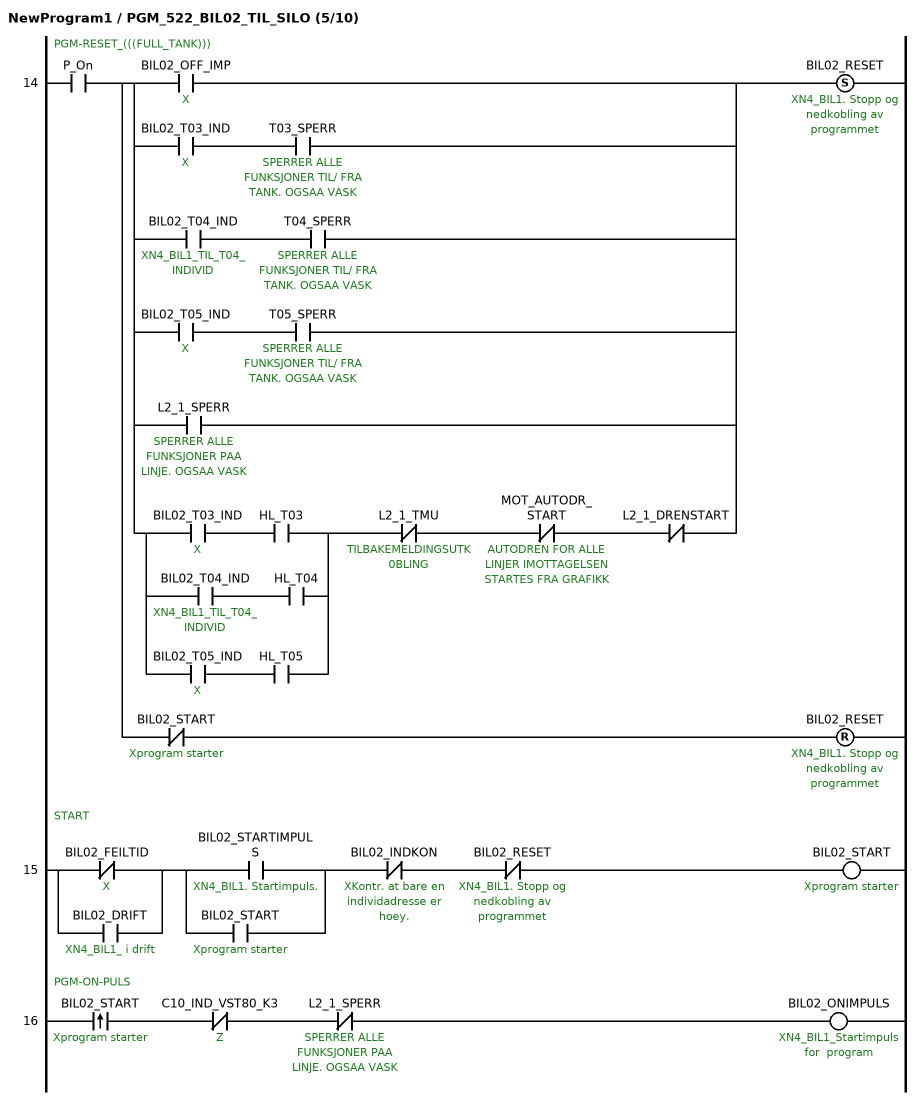
; [picture p624: NewProgram1 / PGM_522_BIL02_TIL_SILO, rungs 14-16]
; rung 14: PGM-RESET_(((FULL_TANK)))
LD P_On
OUT TR0
LD BIL02_OFF_IMP  ; X
LD BIL02_T03_IND  ; X
AND T03_SPERR  ; SPERRER ALLE FUNKSJONER TIL/ FRA TANK. OGSAA VASK
ORLD
LD BIL02_T04_IND  ; XN4_BIL1_TIL_T04_INDIVID
AND T04_SPERR  ; SPERRER ALLE FUNKSJONER TIL/ FRA TANK. OGSAA VASK
ORLD
LD BIL02_T05_IND  ; X
AND T05_SPERR  ; SPERRER ALLE FUNKSJONER TIL/ FRA TANK. OGSAA VASK
ORLD
OR L2_1_SPERR  ; SPERRER ALLE FUNKSJONER PAA LINJE. OGSAA VASK
LD BIL02_T03_IND  ; X
AND HL_T03
LD BIL02_T04_IND  ; XN4_BIL1_TIL_T04_INDIVID
AND HL_T04
ORLD
LD BIL02_T05_IND  ; X
AND HL_T05
ORLD
ANDNOT L2_1_TMU  ; TILBAKEMELDINGSUTK0BLING
ANDNOT MOT_AUTODR_START  ; AUTODREN FOR ALLE LINJER IMOTTAGELSEN STARTES FRA GRAFIKK
ANDNOT L2_1_DRENSTART
ORLD
ANDLD
SET BIL02_RESET  ; XN4_BIL1. Stopp og nedkobling av programmet
LD TR0
ANDNOT BIL02_START  ; Xprogram starter
RSET BIL02_RESET  ; XN4_BIL1. Stopp og nedkobling av programmet
; rung 15: START
LDNOT BIL02_FEILTID  ; X
OR BIL02_DRIFT  ; XN4_BIL1_ i drift
LD BIL02_STARTIMPULS  ; XN4_BIL1. Startimpuls.
OR BIL02_START  ; Xprogram starter
ANDLD
ANDNOT BIL02_INDKON  ; XKontr. at bare en individadresse er hoey.
ANDNOT BIL02_RESET  ; XN4_BIL1. Stopp og nedkobling av programmet
OUT BIL02_START  ; Xprogram starter
; rung 16: PGM-ON-PULS
@LD BIL02_START  ; Xprogram starter
ANDNOT C10_IND_VST80_K3  ; Z
ANDNOT L2_1_SPERR  ; SPERRER ALLE FUNKSJONER PAA LINJE. OGSAA VASK
OUT BIL02_ONIMPULS  ; XN4_BIL1_Startimpuls for  program

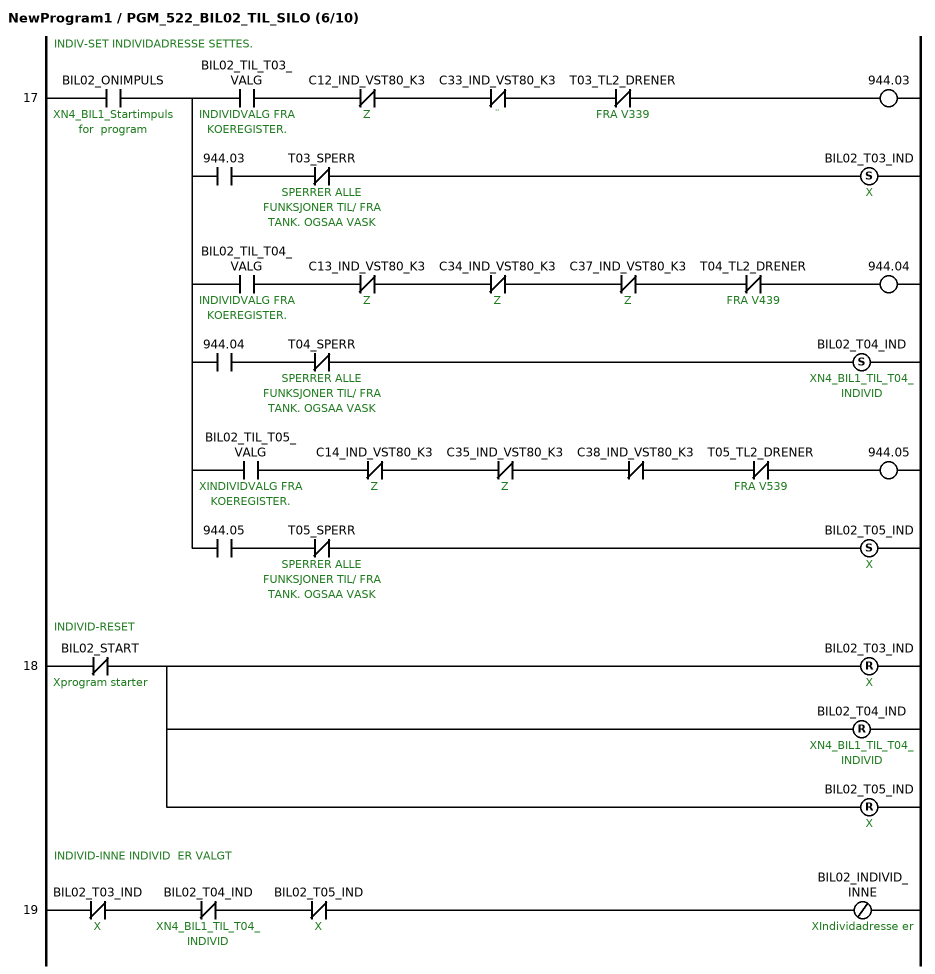
; rung 17: INDIV-SET INDIVIDADRESSE SETTES.
LD BIL02_ONIMPULS  ; XN4_BIL1_Startimpuls for  program
OUT TR0
AND BIL02_TIL_T03_VALG  ; INDIVIDVALG FRA KOEREGISTER.
ANDNOT C12_IND_VST80_K3  ; Z
ANDNOT C33_IND_VST80_K3  ; ¨
ANDNOT T03_TL2_DRENER  ; FRA V339
OUT 944.03
LD TR0
AND 944.03
ANDNOT T03_SPERR  ; SPERRER ALLE FUNKSJONER TIL/ FRA TANK. OGSAA VASK
SET BIL02_T03_IND  ; X
LD TR0
AND BIL02_TIL_T04_VALG  ; INDIVIDVALG FRA KOEREGISTER.
ANDNOT C13_IND_VST80_K3  ; Z
ANDNOT C34_IND_VST80_K3  ; Z
ANDNOT C37_IND_VST80_K3  ; Z
ANDNOT T04_TL2_DRENER  ; FRA V439
OUT 944.04
LD TR0
AND 944.04
ANDNOT T04_SPERR  ; SPERRER ALLE FUNKSJONER TIL/ FRA TANK. OGSAA VASK
SET BIL02_T04_IND  ; XN4_BIL1_TIL_T04_INDIVID
LD TR0
AND BIL02_TIL_T05_VALG  ; XINDIVIDVALG FRA KOEREGISTER.
ANDNOT C14_IND_VST80_K3  ; Z
ANDNOT C35_IND_VST80_K3  ; Z
ANDNOT C38_IND_VST80_K3
ANDNOT T05_TL2_DRENER  ; FRA V539
OUT 944.05
LD TR0
AND 944.05
ANDNOT T05_SPERR  ; SPERRER ALLE FUNKSJONER TIL/ FRA TANK. OGSAA VASK
SET BIL02_T05_IND  ; X
; rung 18: INDIVID-RESET
LDNOT BIL02_START  ; Xprogram starter
RSET BIL02_T03_IND  ; X
RSET BIL02_T04_IND  ; XN4_BIL1_TIL_T04_INDIVID
RSET BIL02_T05_IND  ; X
; rung 19: INDIVID-INNE INDIVID  ER VALGT
LDNOT BIL02_T03_IND  ; X
ANDNOT BIL02_T04_IND  ; XN4_BIL1_TIL_T04_INDIVID
ANDNOT BIL02_T05_IND  ; X
OUTNOT BIL02_INDIVID_INNE  ; XIndividadresse er

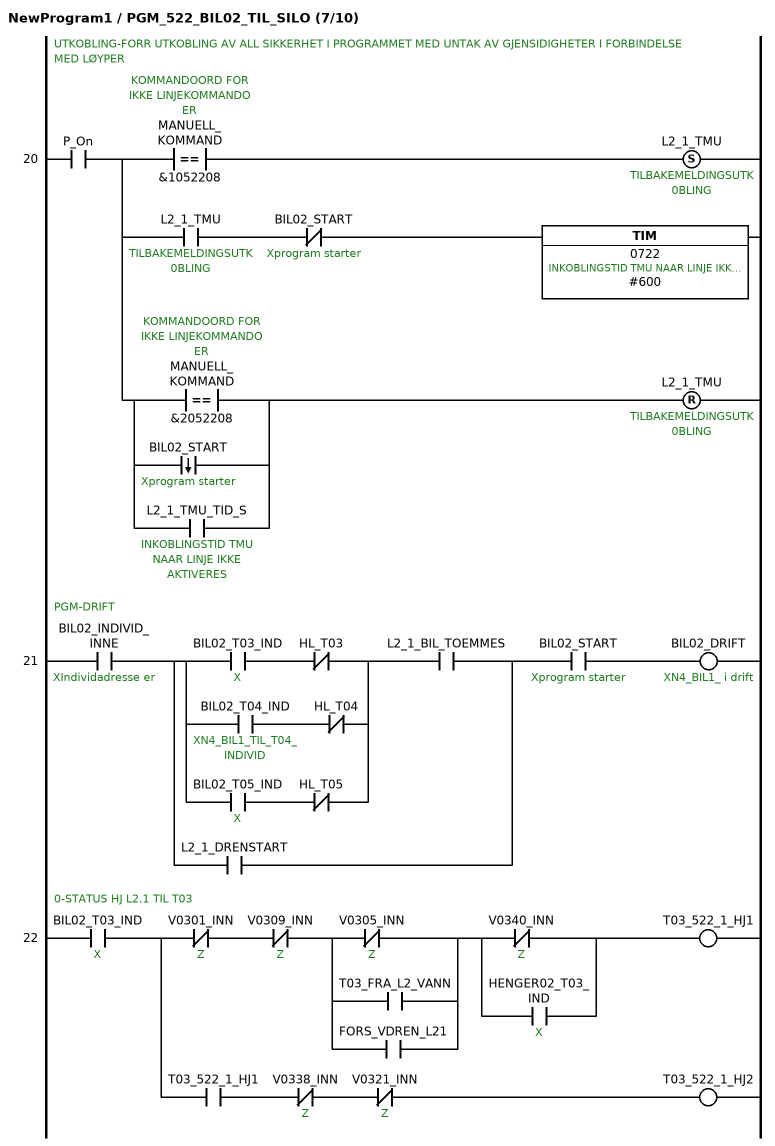
; rung 20: UTKOBLING-FORR UTKOBLING AV ALL SIKKERHET I PROGRAMMET MED UNTAK AV GJENSIDIGHETER I FORBINDELSE MED LØYPER
LD P_On
OUT TR0
AND=L(301) MANUELL_KOMMAND &1052208  ; KOMMANDOORD FOR IKKE LINJEKOMMANDOER
SET L2_1_TMU  ; TILBAKEMELDINGSUTK0BLING
LD TR0
AND L2_1_TMU  ; TILBAKEMELDINGSUTK0BLING
ANDNOT BIL02_START  ; Xprogram starter
TIM 0722 #600  ; INKOBLINGSTID TMU NAAR LINJE IKKE AKTIVERES
LD TR0
LD=L(301) MANUELL_KOMMAND &2052208  ; KOMMANDOORD FOR IKKE LINJEKOMMANDOER
%OR BIL02_START  ; Xprogram starter
OR L2_1_TMU_TID_S  ; INKOBLINGSTID TMU NAAR LINJE IKKE AKTIVERES
ANDLD
RSET L2_1_TMU  ; TILBAKEMELDINGSUTK0BLING
; rung 21: PGM-DRIFT
LD BIL02_INDIVID_INNE  ; XIndividadresse er
LD BIL02_T03_IND  ; X
ANDNOT HL_T03
LD BIL02_T04_IND  ; XN4_BIL1_TIL_T04_INDIVID
ANDNOT HL_T04
ORLD
LD BIL02_T05_IND  ; X
ANDNOT HL_T05
ORLD
AND L2_1_BIL_TOEMMES
OR L2_1_DRENSTART
ANDLD
AND BIL02_START  ; Xprogram starter
OUT BIL02_DRIFT  ; XN4_BIL1_ i drift
; rung 22: 0-STATUS HJ L2.1 TIL T03
LD BIL02_T03_IND  ; X
OUT TR0
ANDNOT V0301_INN  ; Z
ANDNOT V0309_INN  ; Z
LDNOT V0305_INN  ; Z
OR T03_FRA_L2_VANN
OR FORS_VDREN_L21
ANDLD
LDNOT V0340_INN  ; Z
OR HENGER02_T03_IND  ; X
ANDLD
OUT T03_522_1_HJ1
LD TR0
AND T03_522_1_HJ1
ANDNOT V0338_INN  ; Z
ANDNOT V0321_INN  ; Z
OUT T03_522_1_HJ2

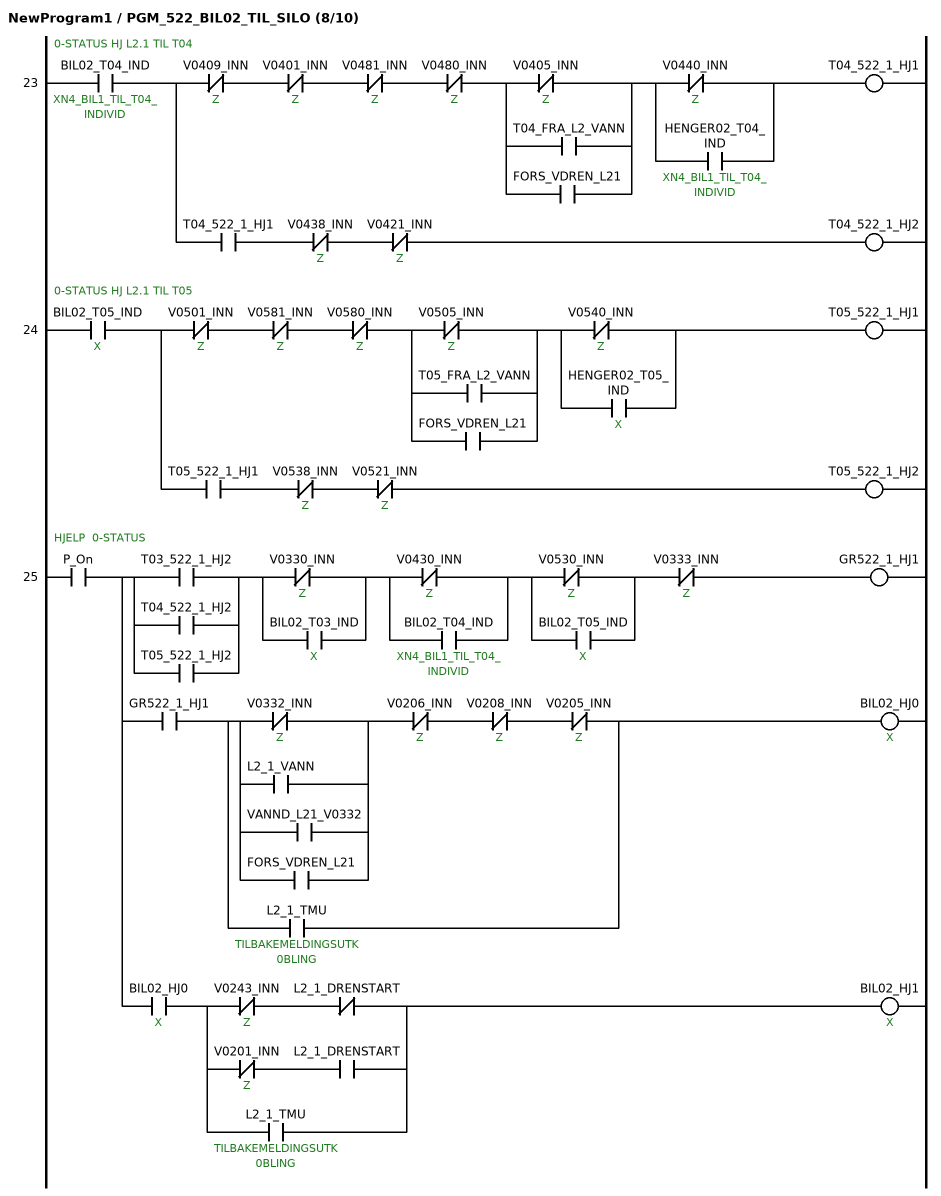
; rung 23: 0-STATUS HJ L2.1 TIL T04
LD BIL02_T04_IND  ; XN4_BIL1_TIL_T04_INDIVID
OUT TR0
ANDNOT V0409_INN  ; Z
ANDNOT V0401_INN  ; Z
ANDNOT V0481_INN  ; Z
ANDNOT V0480_INN  ; Z
LDNOT V0405_INN  ; Z
OR T04_FRA_L2_VANN
OR FORS_VDREN_L21
ANDLD
LDNOT V0440_INN  ; Z
OR HENGER02_T04_IND  ; XN4_BIL1_TIL_T04_INDIVID
ANDLD
OUT T04_522_1_HJ1
LD TR0
AND T04_522_1_HJ1
ANDNOT V0438_INN  ; Z
ANDNOT V0421_INN  ; Z
OUT T04_522_1_HJ2
; rung 24: 0-STATUS HJ L2.1 TIL T05
LD BIL02_T05_IND  ; X
OUT TR0
ANDNOT V0501_INN  ; Z
ANDNOT V0581_INN  ; Z
ANDNOT V0580_INN  ; Z
LDNOT V0505_INN  ; Z
OR T05_FRA_L2_VANN
OR FORS_VDREN_L21
ANDLD
LDNOT V0540_INN  ; Z
OR HENGER02_T05_IND  ; X
ANDLD
OUT T05_522_1_HJ1
LD TR0
AND T05_522_1_HJ1
ANDNOT V0538_INN  ; Z
ANDNOT V0521_INN  ; Z
OUT T05_522_1_HJ2
; rung 25: HJELP  0-STATUS
LD P_On
OUT TR0
LD T03_522_1_HJ2
OR T04_522_1_HJ2
OR T05_522_1_HJ2
ANDLD
LDNOT V0330_INN  ; Z
OR BIL02_T03_IND  ; X
ANDLD
LDNOT V0430_INN  ; Z
OR BIL02_T04_IND  ; XN4_BIL1_TIL_T04_INDIVID
ANDLD
LDNOT V0530_INN  ; Z
OR BIL02_T05_IND  ; X
ANDLD
ANDNOT V0333_INN  ; Z
OUT GR522_1_HJ1
LD TR0
AND GR522_1_HJ1
LDNOT V0332_INN  ; Z
OR L2_1_VANN
OR VANND_L21_V0332
OR FORS_VDREN_L21
ANDNOT V0206_INN  ; Z
ANDNOT V0208_INN  ; Z
ANDNOT V0205_INN  ; Z
OR L2_1_TMU  ; TILBAKEMELDINGSUTK0BLING
ANDLD
OUT BIL02_HJ0  ; X
LD TR0
AND BIL02_HJ0  ; X
LDNOT V0243_INN  ; Z
ANDNOT L2_1_DRENSTART
LDNOT V0201_INN  ; Z
AND L2_1_DRENSTART
ORLD
OR L2_1_TMU  ; TILBAKEMELDINGSUTK0BLING
ANDLD
OUT BIL02_HJ1  ; X

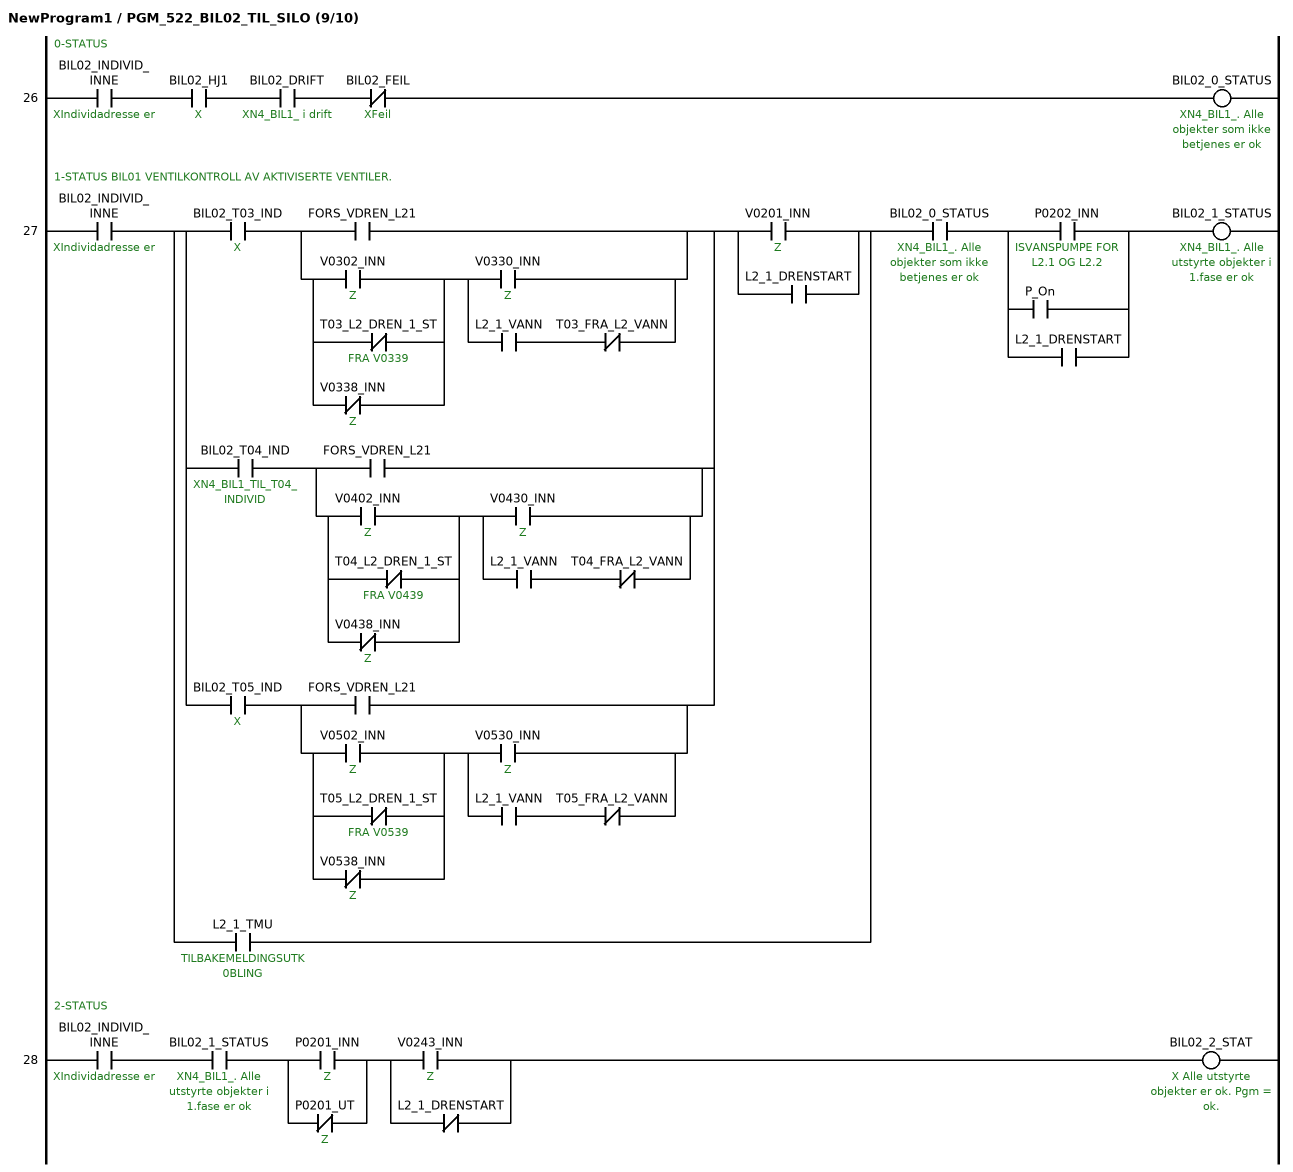
; rung 26: 0-STATUS
LD BIL02_INDIVID_INNE  ; XIndividadresse er
AND BIL02_HJ1  ; X
AND BIL02_DRIFT  ; XN4_BIL1_ i drift
ANDNOT BIL02_FEIL  ; XFeil
OUT BIL02_0_STATUS  ; XN4_BIL1_. Alle objekter som ikke betjenes er ok
; rung 27: 1-STATUS BIL01 VENTILKONTROLL AV AKTIVISERTE VENTILER.
LD BIL02_INDIVID_INNE  ; XIndividadresse er
LD BIL02_T03_IND  ; X
LD FORS_VDREN_L21
LD V0302_INN  ; Z
ORNOT T03_L2_DREN_1_ST  ; FRA V0339
ORNOT V0338_INN  ; Z
LD V0330_INN  ; Z
LD L2_1_VANN
ANDNOT T03_FRA_L2_VANN
ORLD
ANDLD
ORLD
ANDLD
LD BIL02_T04_IND  ; XN4_BIL1_TIL_T04_INDIVID
LD FORS_VDREN_L21
LD V0402_INN  ; Z
ORNOT T04_L2_DREN_1_ST  ; FRA V0439
ORNOT V0438_INN  ; Z
LD V0430_INN  ; Z
LD L2_1_VANN
ANDNOT T04_FRA_L2_VANN
ORLD
ANDLD
ORLD
ANDLD
ORLD
LD BIL02_T05_IND  ; X
LD FORS_VDREN_L21
LD V0502_INN  ; Z
ORNOT T05_L2_DREN_1_ST  ; FRA V0539
ORNOT V0538_INN  ; Z
LD V0530_INN  ; Z
LD L2_1_VANN
ANDNOT T05_FRA_L2_VANN
ORLD
ANDLD
ORLD
ANDLD
ORLD
LD V0201_INN  ; Z
OR L2_1_DRENSTART
ANDLD
OR L2_1_TMU  ; TILBAKEMELDINGSUTK0BLING
ANDLD
AND BIL02_0_STATUS  ; XN4_BIL1_. Alle objekter som ikke betjenes er ok
LD P0202_INN  ; ISVANSPUMPE FOR L2.1 OG L2.2
OR P_On
OR L2_1_DRENSTART
ANDLD
OUT BIL02_1_STATUS  ; XN4_BIL1_. Alle utstyrte objekter i 1.fase er ok
; rung 28: 2-STATUS
LD BIL02_INDIVID_INNE  ; XIndividadresse er
AND BIL02_1_STATUS  ; XN4_BIL1_. Alle utstyrte objekter i 1.fase er ok
LD P0201_INN  ; Z
ORNOT P0201_UT  ; Z
ANDLD
LD V0243_INN  ; Z
ORNOT L2_1_DRENSTART
ANDLD
OUT BIL02_2_STAT  ; X Alle utstyrte objekter er ok. Pgm = ok.

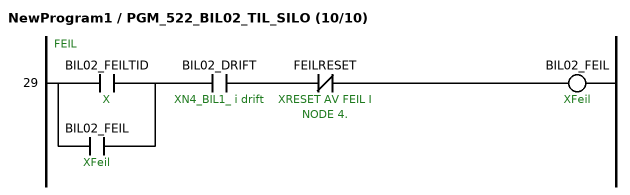
; rung 29: FEIL
LD BIL02_FEILTID  ; X
OR BIL02_FEIL  ; XFeil
AND BIL02_DRIFT  ; XN4_BIL1_ i drift
ANDNOT FEILRESET  ; XRESET AV FEIL I NODE 4.
OUT BIL02_FEIL  ; XFeil
; rung 30: Ingen_kommentar_funnet

### Section V0204_P0201

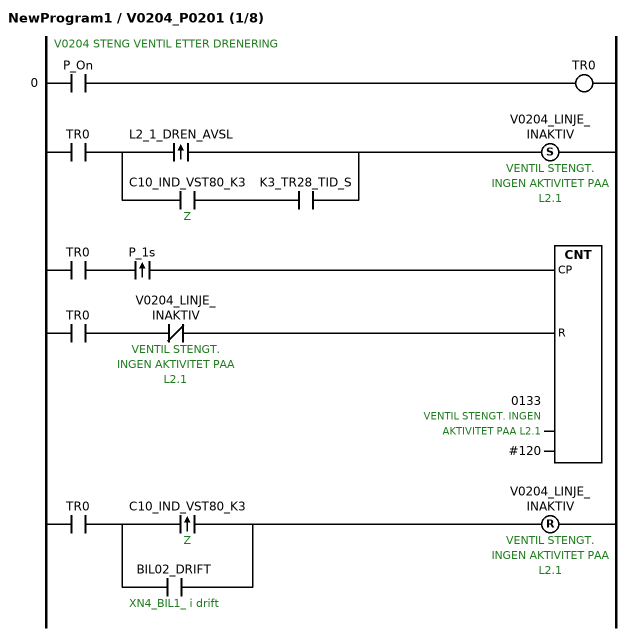
; rung 0: V0204 STENG VENTIL ETTER DRENERING
LD P_On
OUT TR0
@LD L2_1_DREN_AVSL
LD C10_IND_VST80_K3  ; Z
AND K3_TR28_TID_S
ORLD
ANDLD
SET V0204_LINJE_INAKTIV  ; VENTIL STENGT. INGEN AKTIVITET PAA L2.1
LD TR0
@AND P_1s
LD TR0
ANDNOT V0204_LINJE_INAKTIV  ; VENTIL STENGT. INGEN AKTIVITET PAA L2.1
CNT 0133 #120  ; VENTIL STENGT. INGEN AKTIVITET PAA L2.1
LD TR0
@LD C10_IND_VST80_K3  ; Z
OR BIL02_DRIFT  ; XN4_BIL1_ i drift
ANDLD
RSET V0204_LINJE_INAKTIV  ; VENTIL STENGT. INGEN AKTIVITET PAA L2.1

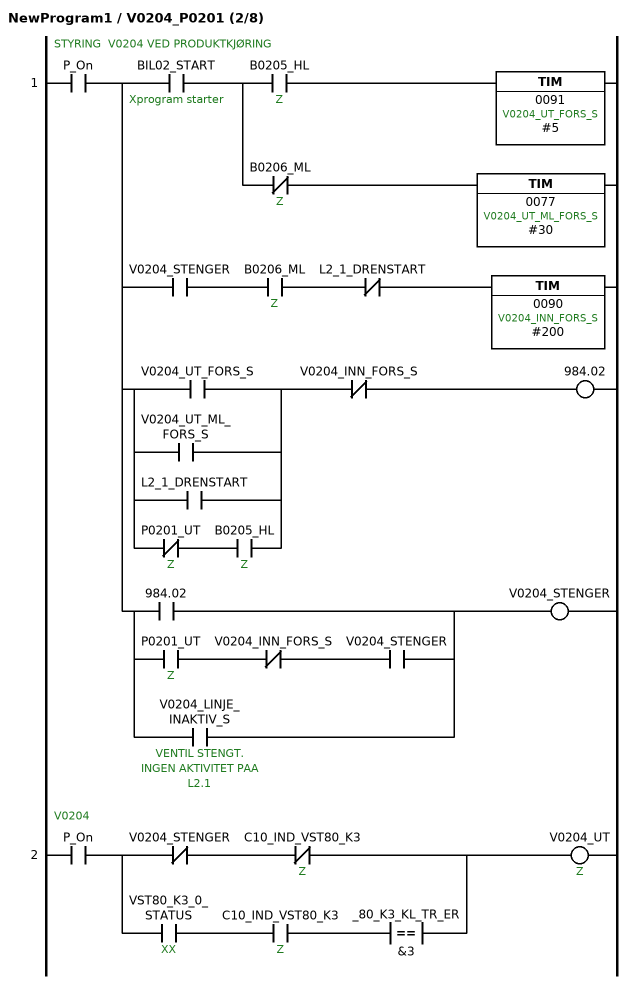
; rung 1: STYRING  V0204 VED PRODUKTKJØRING
LD P_On
OUT TR0
AND BIL02_START  ; Xprogram starter
OUT TR1
AND B0205_HL  ; Z
TIM 0091 #5  ; V0204_UT_FORS_S
LD TR1
ANDNOT B0206_ML  ; Z
TIM 0077 #30  ; V0204_UT_ML_FORS_S
LD TR0
AND V0204_STENGER
AND B0206_ML  ; Z
ANDNOT L2_1_DRENSTART
TIM 0090 #200  ; V0204_INN_FORS_S
LD TR0
LD V0204_UT_FORS_S
OR V0204_UT_ML_FORS_S
OR L2_1_DRENSTART
LDNOT P0201_UT  ; Z
AND B0205_HL  ; Z
ORLD
ANDLD
ANDNOT V0204_INN_FORS_S
OUT 984.02
LD TR0
LD 984.02
LD P0201_UT  ; Z
ANDNOT V0204_INN_FORS_S
AND V0204_STENGER
ORLD
OR V0204_LINJE_INAKTIV_S  ; VENTIL STENGT. INGEN AKTIVITET PAA L2.1
ANDLD
OUT V0204_STENGER
; rung 2: V0204
LD P_On
LDNOT V0204_STENGER
ANDNOT C10_IND_VST80_K3  ; Z
LD VST80_K3_0_STATUS  ; XX
AND C10_IND_VST80_K3  ; Z
AND=(300) _80_K3_KL_TR_ER &3
ORLD
ANDLD
OUT V0204_UT  ; Z

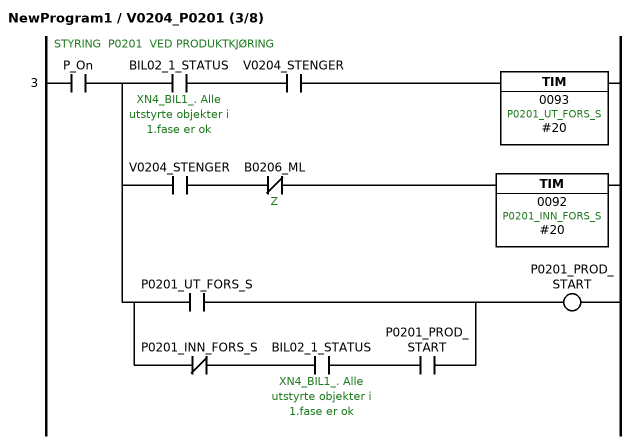
; rung 3: STYRING  P0201  VED PRODUKTKJØRING
LD P_On
OUT TR0
AND BIL02_1_STATUS  ; XN4_BIL1_. Alle utstyrte objekter i 1.fase er ok
AND V0204_STENGER
TIM 0093 #20  ; P0201_UT_FORS_S
LD TR0
AND V0204_STENGER
ANDNOT B0206_ML  ; Z
TIM 0092 #20  ; P0201_INN_FORS_S
LD TR0
LD P0201_UT_FORS_S
LDNOT P0201_INN_FORS_S
AND BIL02_1_STATUS  ; XN4_BIL1_. Alle utstyrte objekter i 1.fase er ok
AND P0201_PROD_START
ORLD
ANDLD
OUT P0201_PROD_START
; rung 4: P0111  ON-OFF STYRING

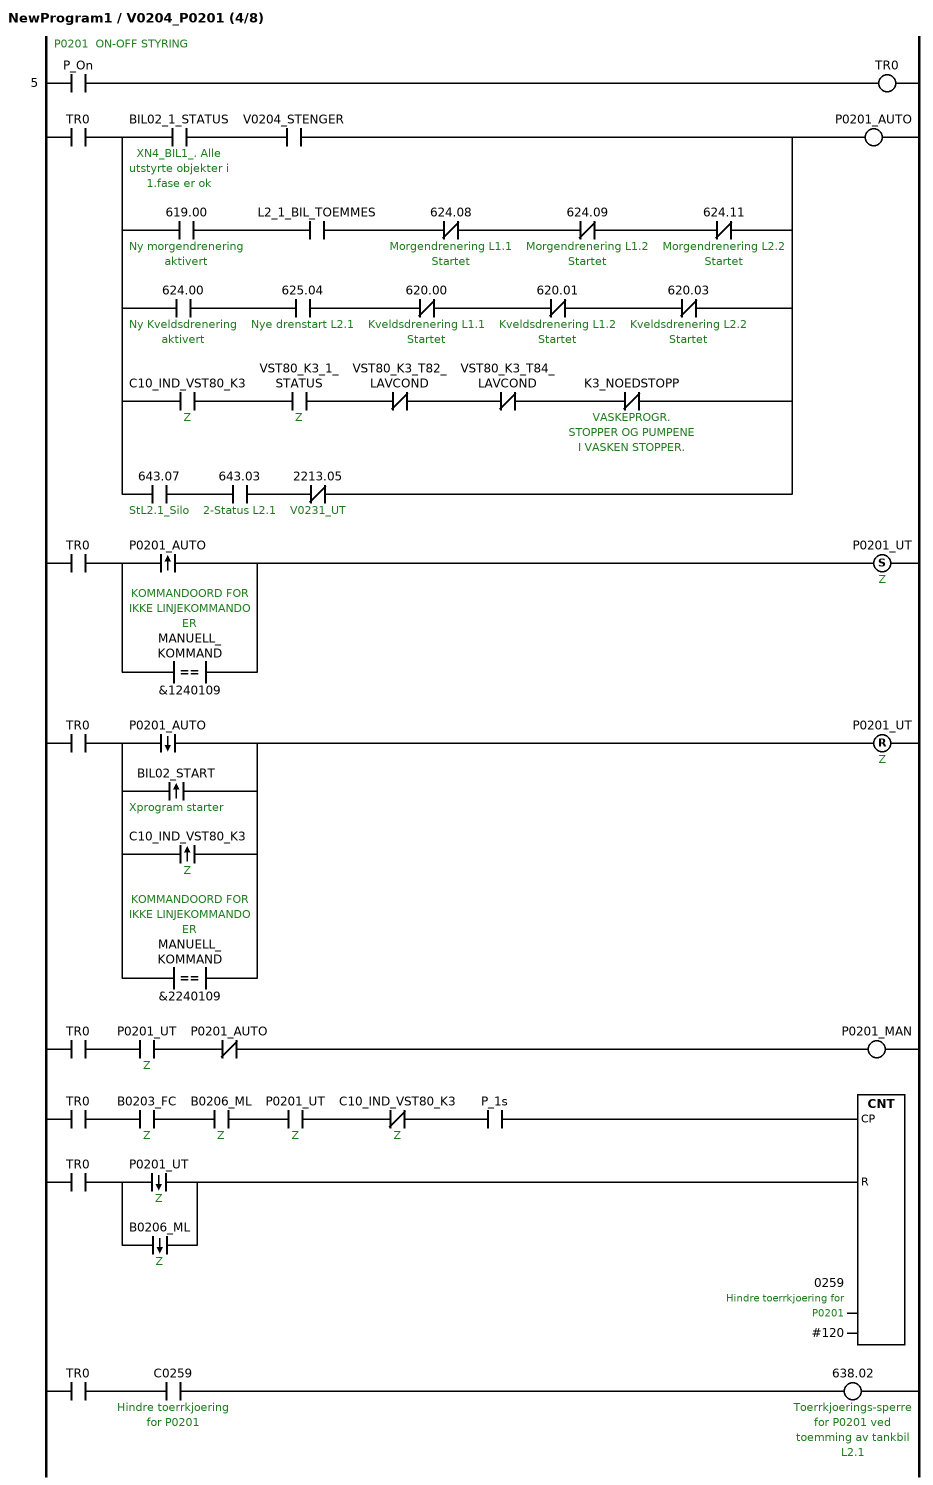
; rung 5: P0201  ON-OFF STYRING
LD P_On
OUT TR0
LD BIL02_1_STATUS  ; XN4_BIL1_. Alle utstyrte objekter i 1.fase er ok
AND V0204_STENGER
LD 619.00  ; Ny morgendrenering aktivert
AND L2_1_BIL_TOEMMES
ANDNOT 624.08  ; Morgendrenering L1.1 Startet
ANDNOT 624.09  ; Morgendrenering L1.2 Startet
ANDNOT 624.11  ; Morgendrenering L2.2 Startet
ORLD
LD 624.00  ; Ny Kveldsdrenering aktivert
AND 625.04  ; Nye drenstart L2.1
ANDNOT 620.00  ; Kveldsdrenering L1.1 Startet
ANDNOT 620.01  ; Kveldsdrenering L1.2 Startet
ANDNOT 620.03  ; Kveldsdrenering L2.2 Startet
ORLD
LD C10_IND_VST80_K3  ; Z
AND VST80_K3_1_STATUS  ; Z
ANDNOT VST80_K3_T82_LAVCOND
ANDNOT VST80_K3_T84_LAVCOND
ANDNOT K3_NOEDSTOPP  ; VASKEPROGR. STOPPER OG PUMPENE I VASKEN STOPPER.
ORLD
LD 643.07  ; StL2.1_Silo
AND 643.03  ; 2-Status L2.1
ANDNOT 2213.05  ; V0231_UT
ORLD
ANDLD
OUT P0201_AUTO
LD TR0
@LD P0201_AUTO
OR=L(301) MANUELL_KOMMAND &1240109  ; KOMMANDOORD FOR IKKE LINJEKOMMANDOER
ANDLD
SET P0201_UT  ; Z
LD TR0
%LD P0201_AUTO
@OR BIL02_START  ; Xprogram starter
@OR C10_IND_VST80_K3  ; Z
OR=L(301) MANUELL_KOMMAND &2240109  ; KOMMANDOORD FOR IKKE LINJEKOMMANDOER
ANDLD
RSET P0201_UT  ; Z
LD TR0
AND P0201_UT  ; Z
ANDNOT P0201_AUTO
OUT P0201_MAN
LD TR0
AND B0203_FC  ; Z
AND B0206_ML  ; Z
AND P0201_UT  ; Z
ANDNOT C10_IND_VST80_K3  ; Z
AND P_1s
LD TR0
%LD P0201_UT  ; Z
%OR B0206_ML  ; Z
ANDLD
CNT 0259 #120  ; Hindre toerrkjoering for P0201
LD TR0
AND C0259  ; Hindre toerrkjoering for P0201
OUT 638.02  ; Toerrkjoerings-sperre for P0201 ved toemming av tankbil L2.1

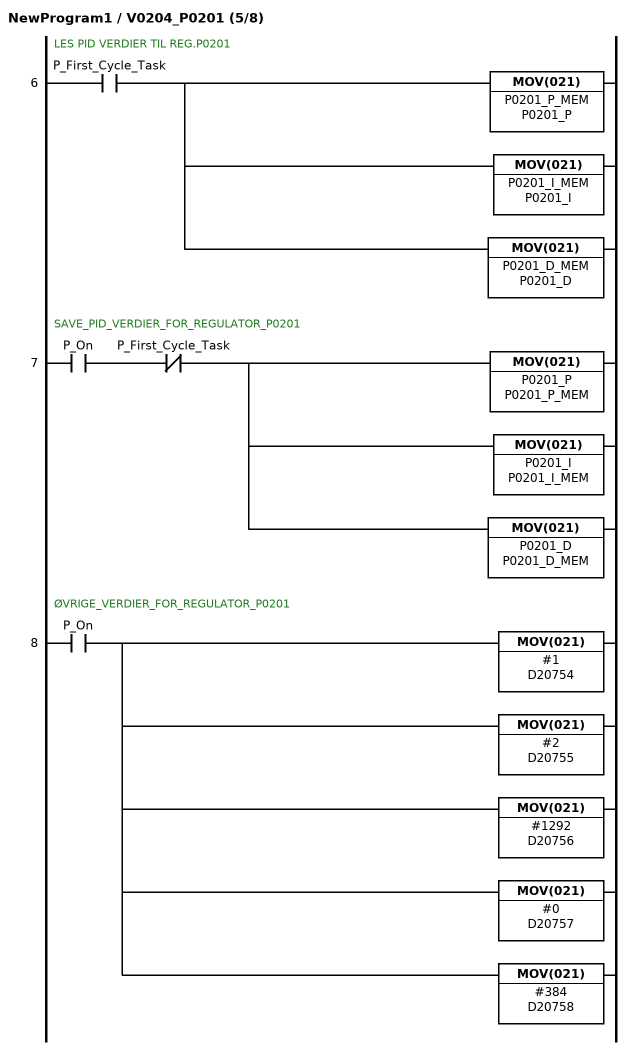
; rung 6: LES PID VERDIER TIL REG.P0201
LD P_First_Cycle_Task
MOV(021) P0201_P_MEM P0201_P
MOV(021) P0201_I_MEM P0201_I
MOV(021) P0201_D_MEM P0201_D
; rung 7: SAVE_PID_VERDIER_FOR_REGULATOR_P0201
LD P_On
ANDNOT P_First_Cycle_Task
MOV(021) P0201_P P0201_P_MEM
MOV(021) P0201_I P0201_I_MEM
MOV(021) P0201_D P0201_D_MEM
; rung 8: ØVRIGE_VERDIER_FOR_REGULATOR_P0201
LD P_On
MOV(021) #1 D20754
MOV(021) #2 D20755
MOV(021) #1292 D20756
MOV(021) #0 D20757
MOV(021) #384 D20758

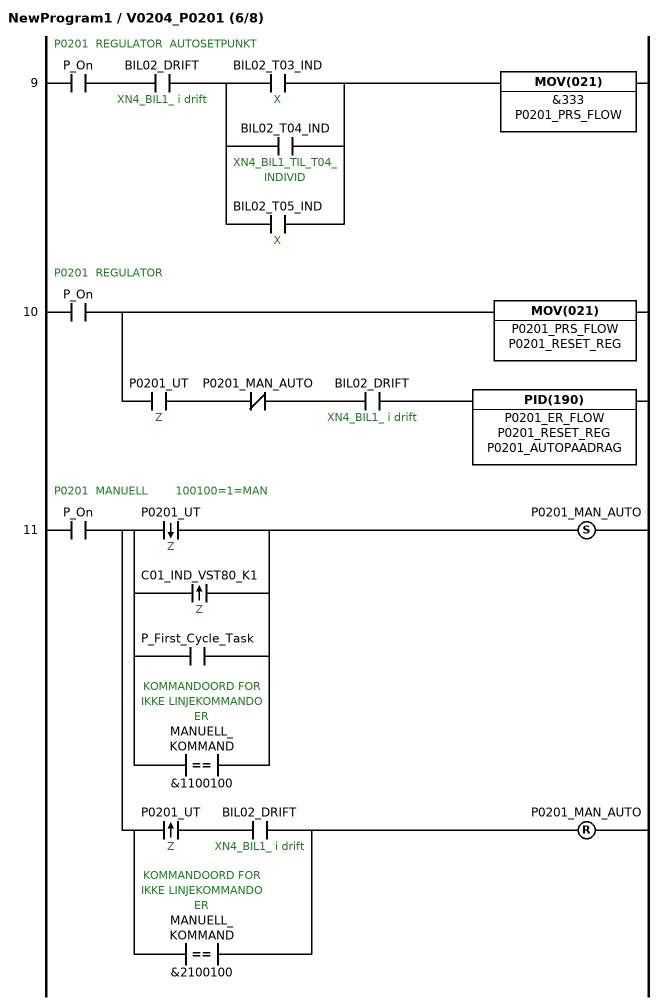
; rung 9: P0201  REGULATOR  AUTOSETPUNKT
LD P_On
AND BIL02_DRIFT  ; XN4_BIL1_ i drift
LD BIL02_T03_IND  ; X
OR BIL02_T04_IND  ; XN4_BIL1_TIL_T04_INDIVID
OR BIL02_T05_IND  ; X
ANDLD
MOV(021) &333 P0201_PRS_FLOW
; rung 10: P0201  REGULATOR
LD P_On
MOV(021) P0201_PRS_FLOW P0201_RESET_REG
AND P0201_UT  ; Z
ANDNOT P0201_MAN_AUTO
AND BIL02_DRIFT  ; XN4_BIL1_ i drift
PID(190) P0201_ER_FLOW P0201_RESET_REG P0201_AUTOPAADRAG
; rung 11: P0201  MANUELL        100100=1=MAN
LD P_On
OUT TR0
%LD P0201_UT  ; Z
@OR C01_IND_VST80_K1  ; Z
OR P_First_Cycle_Task
OR=L(301) MANUELL_KOMMAND &1100100  ; KOMMANDOORD FOR IKKE LINJEKOMMANDOER
ANDLD
SET P0201_MAN_AUTO
LD TR0
@LD P0201_UT  ; Z
AND BIL02_DRIFT  ; XN4_BIL1_ i drift
OR=L(301) MANUELL_KOMMAND &2100100  ; KOMMANDOORD FOR IKKE LINJEKOMMANDOER
ANDLD
RSET P0201_MAN_AUTO

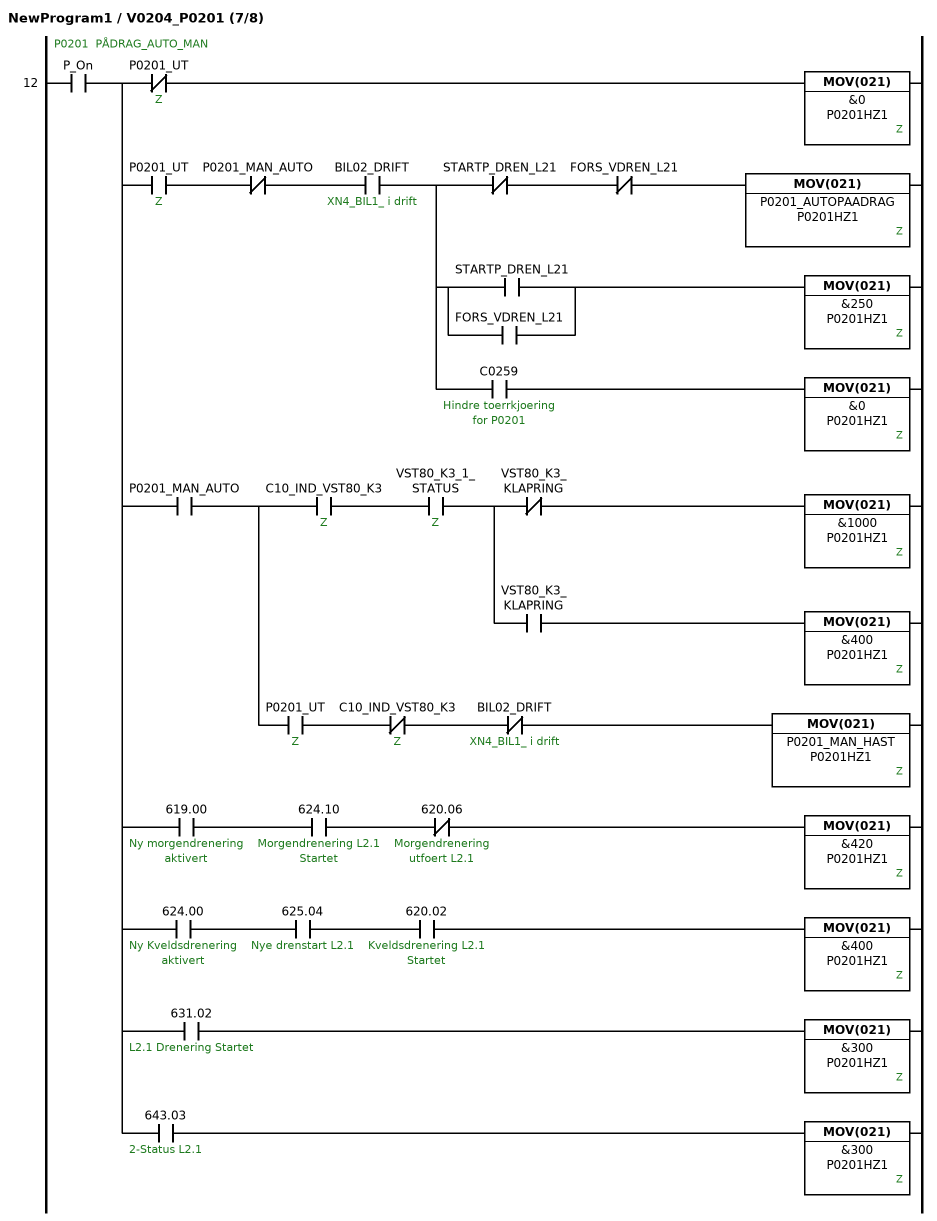
; rung 12: P0201  PÅDRAG_AUTO_MAN
LD P_On
OUT TR0
ANDNOT P0201_UT  ; Z
MOV(021) &0 P0201HZ1  ; Z
LD TR0
AND P0201_UT  ; Z
ANDNOT P0201_MAN_AUTO
AND BIL02_DRIFT  ; XN4_BIL1_ i drift
OUT TR1
ANDNOT STARTP_DREN_L21
ANDNOT FORS_VDREN_L21
MOV(021) P0201_AUTOPAADRAG P0201HZ1  ; Z
LD TR1
LD STARTP_DREN_L21
OR FORS_VDREN_L21
ANDLD
MOV(021) &250 P0201HZ1  ; Z
LD TR1
AND C0259  ; Hindre toerrkjoering for P0201
MOV(021) &0 P0201HZ1  ; Z
LD TR0
AND P0201_MAN_AUTO
OUT TR1
AND C10_IND_VST80_K3  ; Z
AND VST80_K3_1_STATUS  ; Z
OUT TR2
ANDNOT VST80_K3_KLAPRING
MOV(021) &1000 P0201HZ1  ; Z
LD TR2
AND VST80_K3_KLAPRING
MOV(021) &400 P0201HZ1  ; Z
LD TR1
AND P0201_UT  ; Z
ANDNOT C10_IND_VST80_K3  ; Z
ANDNOT BIL02_DRIFT  ; XN4_BIL1_ i drift
MOV(021) P0201_MAN_HAST P0201HZ1  ; Z
LD TR0
AND 619.00  ; Ny morgendrenering aktivert
AND 624.10  ; Morgendrenering L2.1 Startet
ANDNOT 620.06  ; Morgendrenering utfoert L2.1
MOV(021) &420 P0201HZ1  ; Z
LD TR0
AND 624.00  ; Ny Kveldsdrenering aktivert
AND 625.04  ; Nye drenstart L2.1
AND 620.02  ; Kveldsdrenering L2.1 Startet
MOV(021) &400 P0201HZ1  ; Z
LD TR0
AND 631.02  ; L2.1 Drenering Startet
MOV(021) &300 P0201HZ1  ; Z
LD TR0
AND 643.03  ; 2-Status L2.1
MOV(021) &300 P0201HZ1  ; Z

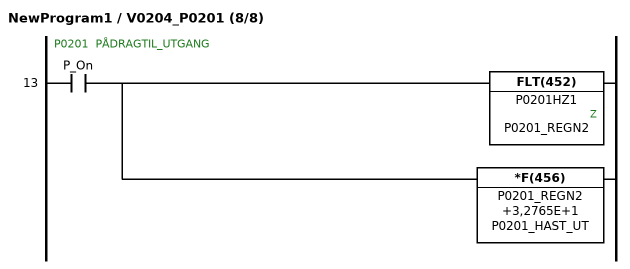
; rung 13: P0201  PÅDRAGTIL_UTGANG
LD P_On
FLT(452) P0201HZ1 P0201_REGN2  ; Z
*F(456) P0201_REGN2 +3,2765E+1 P0201_HAST_UT
; rung 14: Ingen_kommentar_funnet

### Section P0202_ISVANN

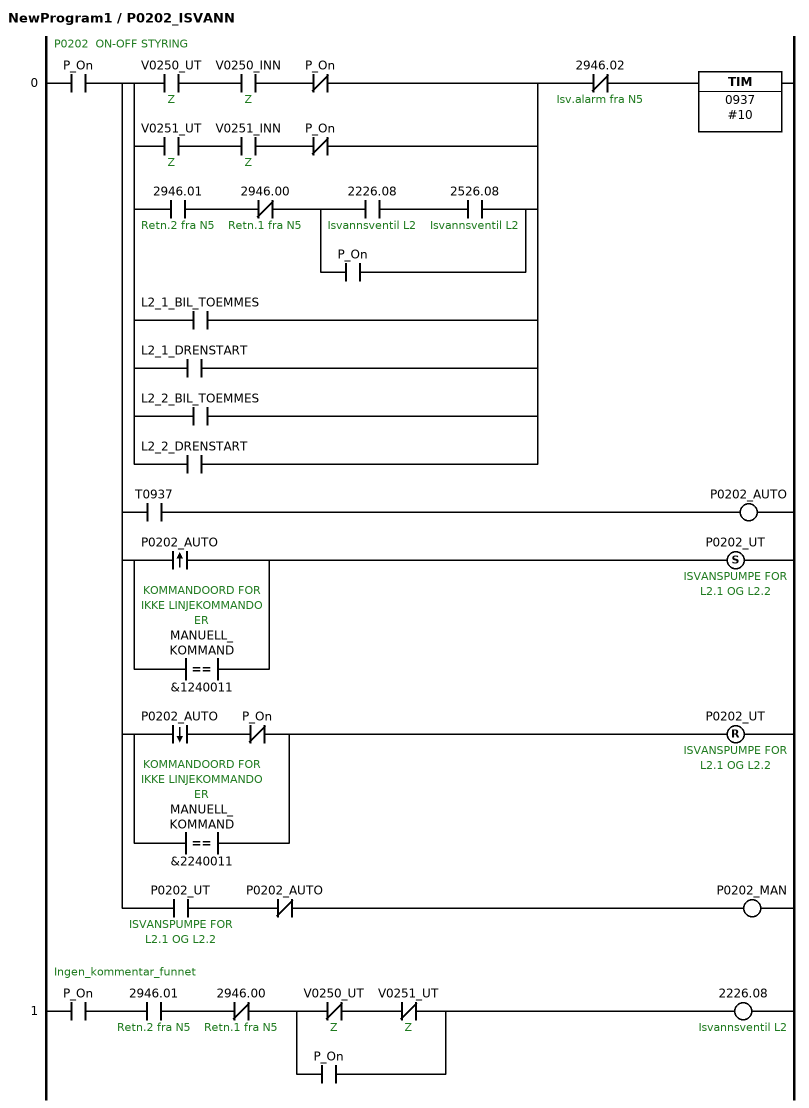
; rung 0: P0202  ON-OFF STYRING
LD P_On
OUT TR0
LD V0250_UT  ; Z
AND V0250_INN  ; Z
ANDNOT P_On
LD V0251_UT  ; Z
AND V0251_INN  ; Z
ANDNOT P_On
ORLD
LD 2946.01  ; Retn.2 fra N5
ANDNOT 2946.00  ; Retn.1 fra N5
LD 2226.08  ; Isvannsventil L2
AND 2526.08  ; Isvannsventil L2
OR P_On
ANDLD
ORLD
OR L2_1_BIL_TOEMMES
OR L2_1_DRENSTART
OR L2_2_BIL_TOEMMES
OR L2_2_DRENSTART
ANDLD
ANDNOT 2946.02  ; Isv.alarm fra N5
TIM 0937 #10
LD TR0
AND T0937
OUT P0202_AUTO
LD TR0
@LD P0202_AUTO
OR=L(301) MANUELL_KOMMAND &1240011  ; KOMMANDOORD FOR IKKE LINJEKOMMANDOER
ANDLD
SET P0202_UT  ; ISVANSPUMPE FOR L2.1 OG L2.2
LD TR0
%LD P0202_AUTO
ANDNOT P_On
OR=L(301) MANUELL_KOMMAND &2240011  ; KOMMANDOORD FOR IKKE LINJEKOMMANDOER
ANDLD
RSET P0202_UT  ; ISVANSPUMPE FOR L2.1 OG L2.2
LD TR0
AND P0202_UT  ; ISVANSPUMPE FOR L2.1 OG L2.2
ANDNOT P0202_AUTO
OUT P0202_MAN
; rung 1: Ingen_kommentar_funnet
LD P_On
AND 2946.01  ; Retn.2 fra N5
ANDNOT 2946.00  ; Retn.1 fra N5
LDNOT V0250_UT  ; Z
ANDNOT V0251_UT  ; Z
OR P_On
ANDLD
OUT 2226.08  ; Isvannsventil L2
; rung 2: Ingen_kommentar_funnet

### Section V0250_V0253_ISV

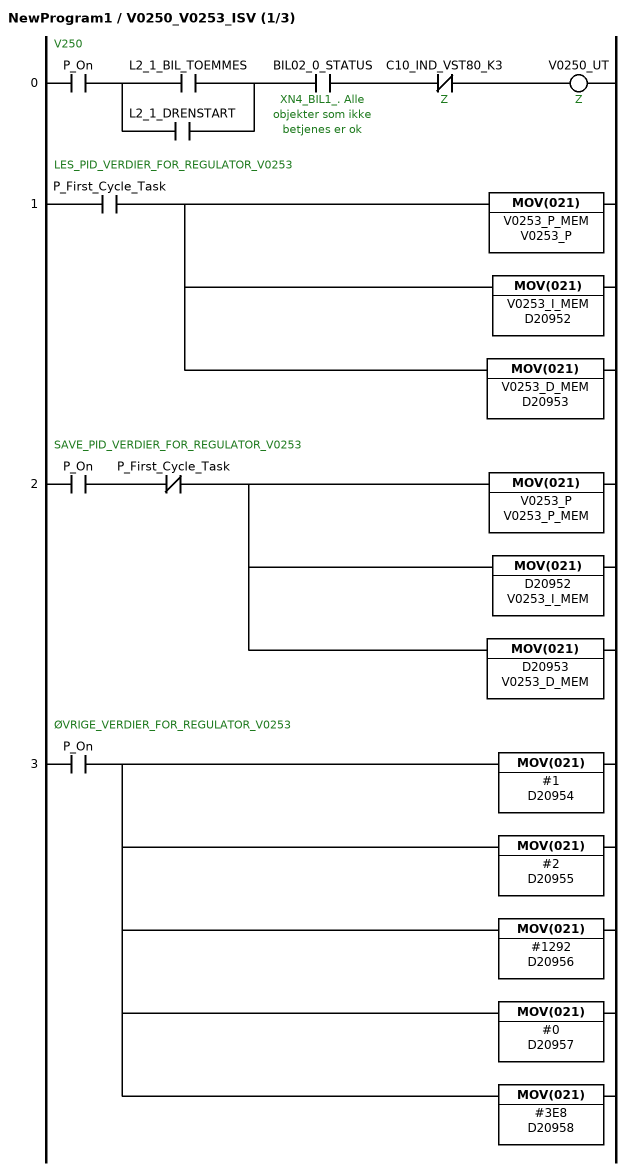
; rung 0: V250
LD P_On
LD L2_1_BIL_TOEMMES
OR L2_1_DRENSTART
ANDLD
AND BIL02_0_STATUS  ; XN4_BIL1_. Alle objekter som ikke betjenes er ok
ANDNOT C10_IND_VST80_K3  ; Z
OUT V0250_UT  ; Z
; rung 1: LES_PID_VERDIER_FOR_REGULATOR_V0253
LD P_First_Cycle_Task
MOV(021) V0253_P_MEM V0253_P
MOV(021) V0253_I_MEM D20952
MOV(021) V0253_D_MEM D20953
; rung 2: SAVE_PID_VERDIER_FOR_REGULATOR_V0253
LD P_On
ANDNOT P_First_Cycle_Task
MOV(021) V0253_P V0253_P_MEM
MOV(021) D20952 V0253_I_MEM
MOV(021) D20953 V0253_D_MEM
; rung 3: ØVRIGE_VERDIER_FOR_REGULATOR_V0253
LD P_On
MOV(021) #1 D20954
MOV(021) #2 D20955
MOV(021) #1292 D20956
MOV(021) #0 D20957
MOV(021) #3E8 D20958

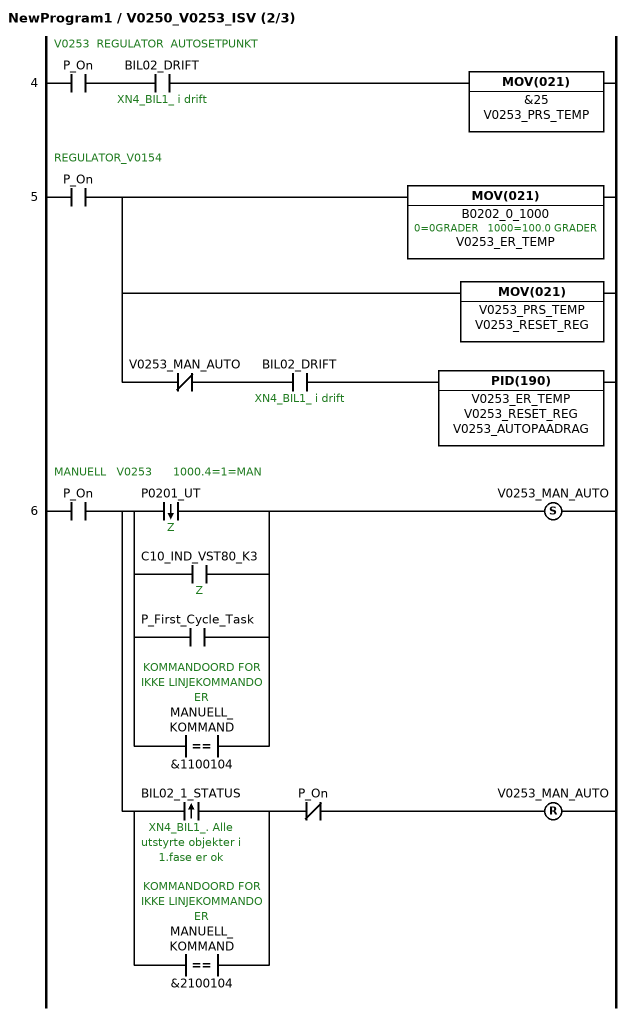
; rung 4: V0253  REGULATOR  AUTOSETPUNKT
LD P_On
AND BIL02_DRIFT  ; XN4_BIL1_ i drift
MOV(021) &25 V0253_PRS_TEMP
; rung 5: REGULATOR_V0154
LD P_On
MOV(021) B0202_0_1000 V0253_ER_TEMP  ; 0=0GRADER   1000=100.0 GRADER
MOV(021) V0253_PRS_TEMP V0253_RESET_REG
ANDNOT V0253_MAN_AUTO
AND BIL02_DRIFT  ; XN4_BIL1_ i drift
PID(190) V0253_ER_TEMP V0253_RESET_REG V0253_AUTOPAADRAG
; rung 6: MANUELL   V0253      1000.4=1=MAN
LD P_On
OUT TR0
%LD P0201_UT  ; Z
OR C10_IND_VST80_K3  ; Z
OR P_First_Cycle_Task
OR=L(301) MANUELL_KOMMAND &1100104  ; KOMMANDOORD FOR IKKE LINJEKOMMANDOER
ANDLD
SET V0253_MAN_AUTO
LD TR0
@LD BIL02_1_STATUS  ; XN4_BIL1_. Alle utstyrte objekter i 1.fase er ok
OR=L(301) MANUELL_KOMMAND &2100104  ; KOMMANDOORD FOR IKKE LINJEKOMMANDOER
ANDLD
ANDNOT P_On
RSET V0253_MAN_AUTO

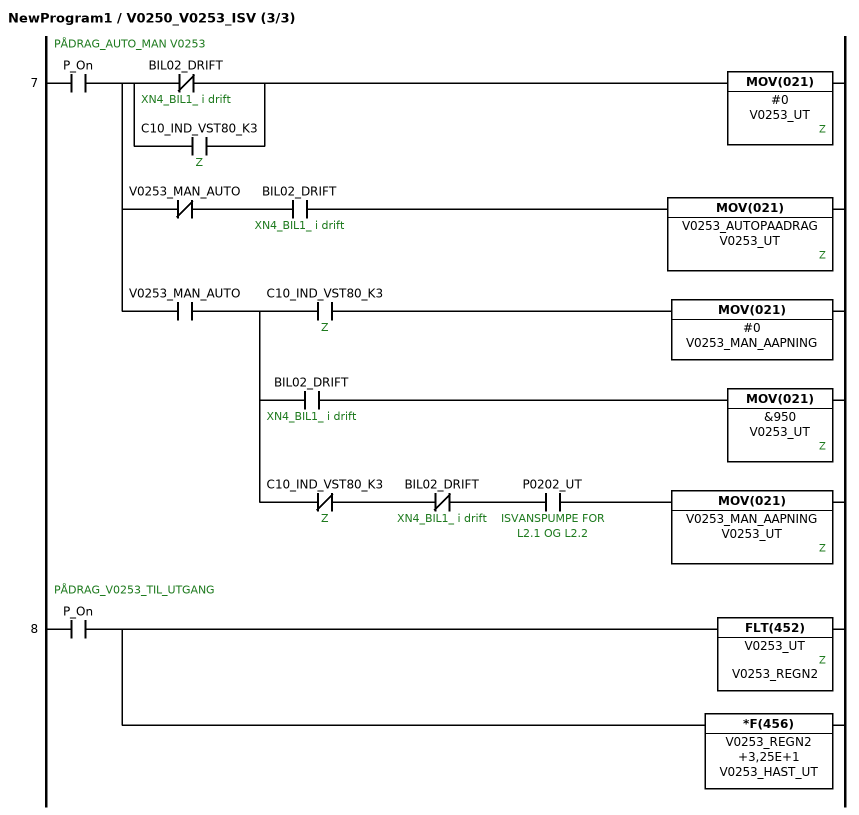
; rung 7: PÅDRAG_AUTO_MAN V0253
LD P_On
OUT TR0
LDNOT BIL02_DRIFT  ; XN4_BIL1_ i drift
OR C10_IND_VST80_K3  ; Z
ANDLD
MOV(021) #0 V0253_UT  ; Z
LD TR0
ANDNOT V0253_MAN_AUTO
AND BIL02_DRIFT  ; XN4_BIL1_ i drift
MOV(021) V0253_AUTOPAADRAG V0253_UT  ; Z
LD TR0
AND V0253_MAN_AUTO
OUT TR0
AND C10_IND_VST80_K3  ; Z
MOV(021) #0 V0253_MAN_AAPNING
LD TR0
AND BIL02_DRIFT  ; XN4_BIL1_ i drift
MOV(021) &950 V0253_UT  ; Z
LD TR0
ANDNOT C10_IND_VST80_K3  ; Z
ANDNOT BIL02_DRIFT  ; XN4_BIL1_ i drift
AND P0202_UT  ; ISVANSPUMPE FOR L2.1 OG L2.2
MOV(021) V0253_MAN_AAPNING V0253_UT  ; Z
; rung 8: PÅDRAG_V0253_TIL_UTGANG
LD P_On
FLT(452) V0253_UT V0253_REGN2  ; Z
*F(456) V0253_REGN2 +3,25E+1 V0253_HAST_UT
; rung 9: Ingen_kommentar_funnet

### Section PGM_523_HENGER02_TIL_SILO

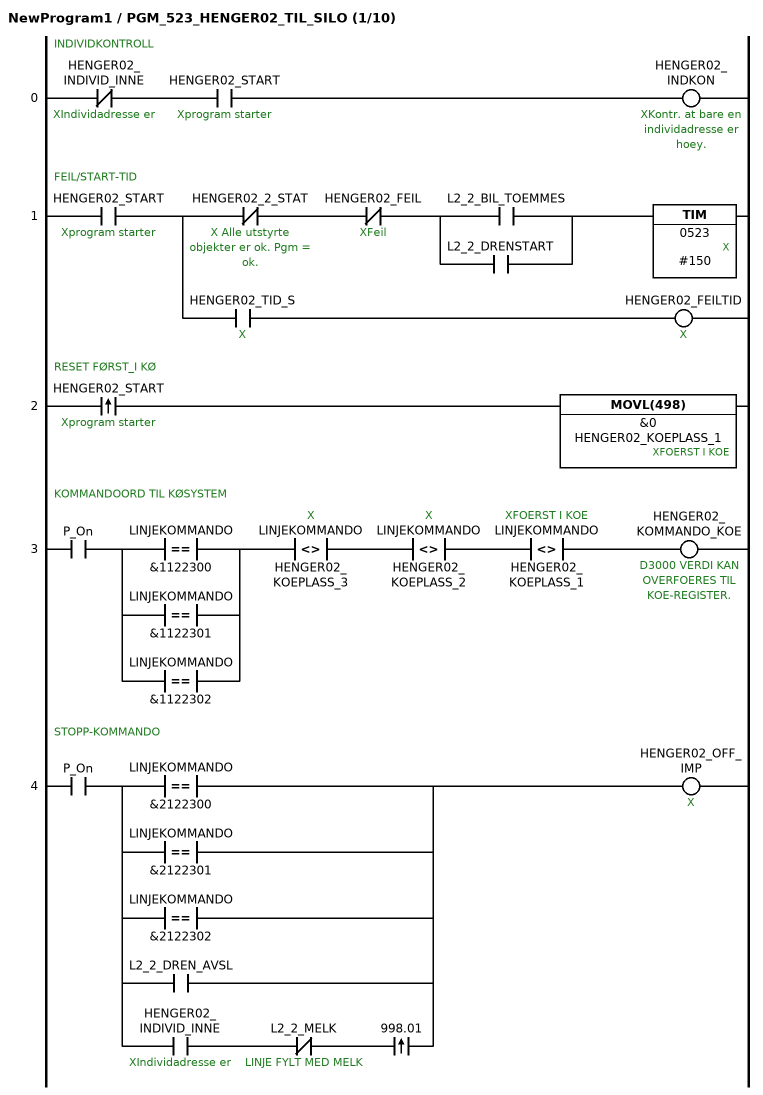
; rung 0: INDIVIDKONTROLL
LDNOT HENGER02_INDIVID_INNE  ; XIndividadresse er
AND HENGER02_START  ; Xprogram starter
OUT HENGER02_INDKON  ; XKontr. at bare en individadresse er hoey.
; rung 1: FEIL/START-TID
LD HENGER02_START  ; Xprogram starter
OUT TR0
ANDNOT HENGER02_2_STAT  ; X Alle utstyrte objekter er ok. Pgm = ok.
ANDNOT HENGER02_FEIL  ; XFeil
LD L2_2_BIL_TOEMMES
OR L2_2_DRENSTART
ANDLD
TIM 0523 #150  ; X
LD TR0
AND HENGER02_TID_S  ; X
OUT HENGER02_FEILTID  ; X
; rung 2: RESET FØRST_I KØ
@LD HENGER02_START  ; Xprogram starter
MOVL(498) &0 HENGER02_KOEPLASS_1  ; XFOERST I KOE
; rung 3: KOMMANDOORD TIL KØSYSTEM
LD P_On
LD=L(301) LINJEKOMMANDO &1122300
OR=L(301) LINJEKOMMANDO &1122301
OR=L(301) LINJEKOMMANDO &1122302
ANDLD
AND<>L(306) LINJEKOMMANDO HENGER02_KOEPLASS_3  ; X
AND<>L(306) LINJEKOMMANDO HENGER02_KOEPLASS_2  ; X
AND<>L(306) LINJEKOMMANDO HENGER02_KOEPLASS_1  ; XFOERST I KOE
OUT HENGER02_KOMMANDO_KOE  ; D3000 VERDI KAN OVERFOERES TIL KOE-REGISTER.
; rung 4: STOPP-KOMMANDO
LD P_On
LD=L(301) LINJEKOMMANDO &2122300
OR=L(301) LINJEKOMMANDO &2122301
OR=L(301) LINJEKOMMANDO &2122302
OR L2_2_DREN_AVSL
LD HENGER02_INDIVID_INNE  ; XIndividadresse er
ANDNOT L2_2_MELK  ; LINJE FYLT MED MELK
@AND 998.01
ORLD
ANDLD
OUT HENGER02_OFF_IMP  ; X

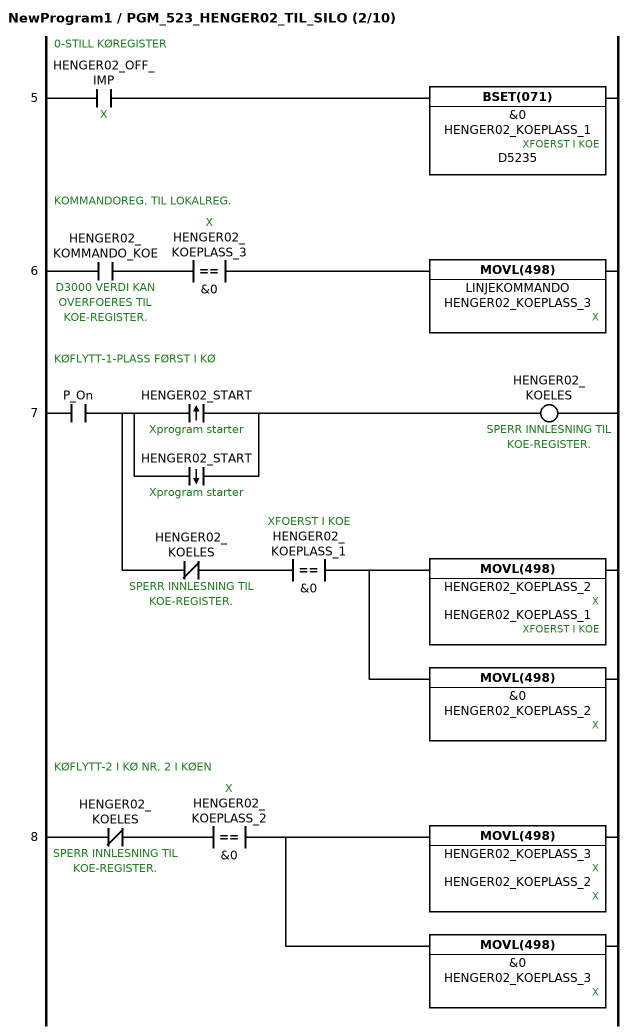
; rung 5: 0-STILL KØREGISTER
LD HENGER02_OFF_IMP  ; X
BSET(071) &0 HENGER02_KOEPLASS_1 D5235  ; XFOERST I KOE
; rung 6: KOMMANDOREG. TIL LOKALREG.
LD HENGER02_KOMMANDO_KOE  ; D3000 VERDI KAN OVERFOERES TIL KOE-REGISTER.
AND=L(301) HENGER02_KOEPLASS_3 &0  ; X
MOVL(498) LINJEKOMMANDO HENGER02_KOEPLASS_3  ; X
; rung 7: KØFLYTT-1-PLASS FØRST I KØ
LD P_On
OUT TR0
@LD HENGER02_START  ; Xprogram starter
%OR HENGER02_START  ; Xprogram starter
ANDLD
OUT HENGER02_KOELES  ; SPERR INNLESNING TIL KOE-REGISTER.
LD TR0
ANDNOT HENGER02_KOELES  ; SPERR INNLESNING TIL KOE-REGISTER.
AND=L(301) HENGER02_KOEPLASS_1 &0  ; XFOERST I KOE
MOVL(498) HENGER02_KOEPLASS_2 HENGER02_KOEPLASS_1  ; X, XFOERST I KOE
MOVL(498) &0 HENGER02_KOEPLASS_2  ; X
; rung 8: KØFLYTT-2 I KØ NR. 2 I KØEN
LDNOT HENGER02_KOELES  ; SPERR INNLESNING TIL KOE-REGISTER.
AND=L(301) HENGER02_KOEPLASS_2 &0  ; X
MOVL(498) HENGER02_KOEPLASS_3 HENGER02_KOEPLASS_2  ; X
MOVL(498) &0 HENGER02_KOEPLASS_3  ; X

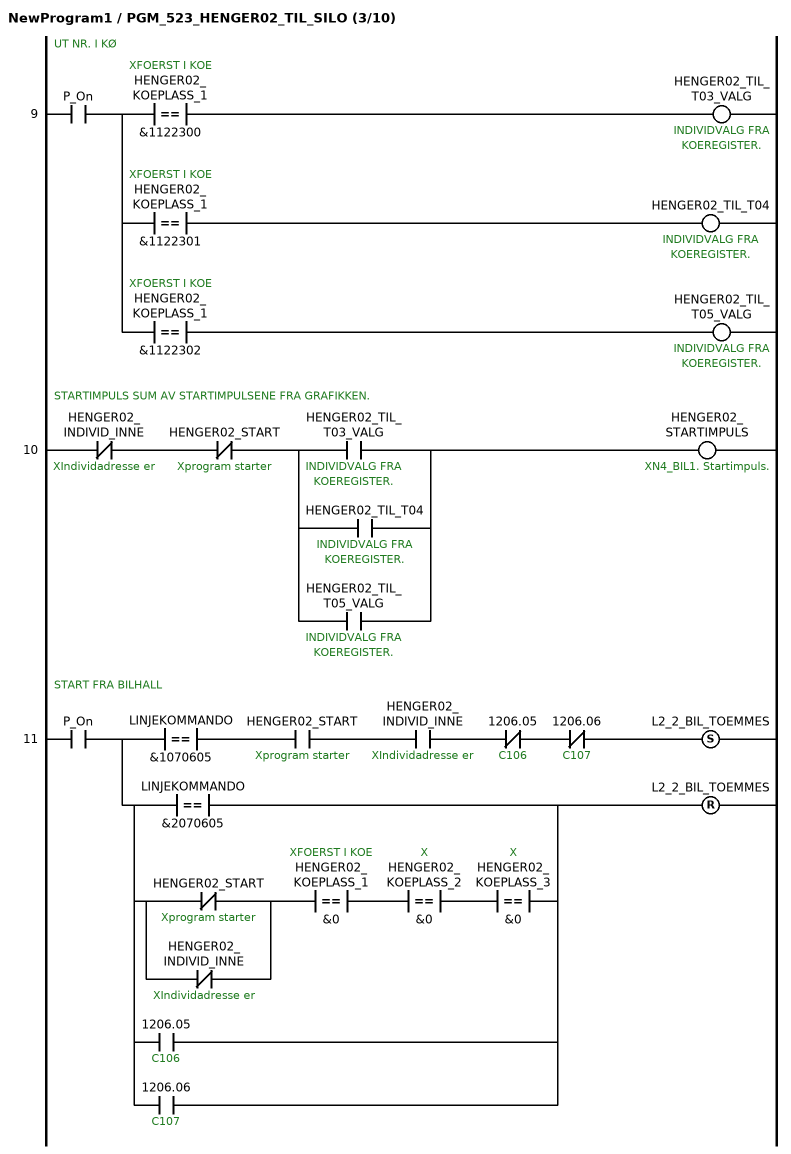
; rung 9: UT NR. I KØ
LD P_On
OUT TR0
AND=L(301) HENGER02_KOEPLASS_1 &1122300  ; XFOERST I KOE
OUT HENGER02_TIL_T03_VALG  ; INDIVIDVALG FRA KOEREGISTER.
LD TR0
AND=L(301) HENGER02_KOEPLASS_1 &1122301  ; XFOERST I KOE
OUT HENGER02_TIL_T04  ; INDIVIDVALG FRA KOEREGISTER.
LD TR0
AND=L(301) HENGER02_KOEPLASS_1 &1122302  ; XFOERST I KOE
OUT HENGER02_TIL_T05_VALG  ; INDIVIDVALG FRA KOEREGISTER.
; rung 10: STARTIMPULS SUM AV STARTIMPULSENE FRA GRAFIKKEN.
LDNOT HENGER02_INDIVID_INNE  ; XIndividadresse er
ANDNOT HENGER02_START  ; Xprogram starter
LD HENGER02_TIL_T03_VALG  ; INDIVIDVALG FRA KOEREGISTER.
OR HENGER02_TIL_T04  ; INDIVIDVALG FRA KOEREGISTER.
OR HENGER02_TIL_T05_VALG  ; INDIVIDVALG FRA KOEREGISTER.
ANDLD
OUT HENGER02_STARTIMPULS  ; XN4_BIL1. Startimpuls.
; rung 11: START FRA BILHALL
LD P_On
OUT TR0
AND=L(301) LINJEKOMMANDO &1070605
AND HENGER02_START  ; Xprogram starter
AND HENGER02_INDIVID_INNE  ; XIndividadresse er
ANDNOT 1206.05  ; C106
ANDNOT 1206.06  ; C107
SET L2_2_BIL_TOEMMES
LD TR0
LD=L(301) LINJEKOMMANDO &2070605
LDNOT HENGER02_START  ; Xprogram starter
ORNOT HENGER02_INDIVID_INNE  ; XIndividadresse er
AND=(300) HENGER02_KOEPLASS_1 &0  ; XFOERST I KOE
AND=(300) HENGER02_KOEPLASS_2 &0  ; X
AND=(300) HENGER02_KOEPLASS_3 &0  ; X
ORLD
OR 1206.05  ; C106
OR 1206.06  ; C107
ANDLD
RSET L2_2_BIL_TOEMMES

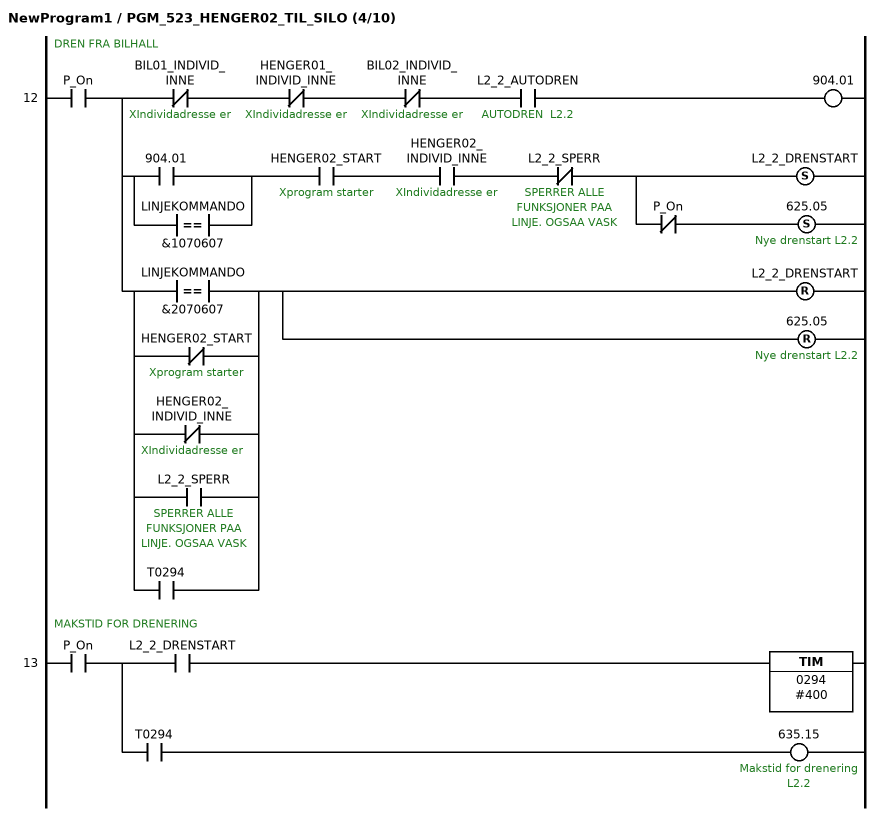
; rung 12: DREN FRA BILHALL
LD P_On
OUT TR0
ANDNOT BIL01_INDIVID_INNE  ; XIndividadresse er
ANDNOT HENGER01_INDIVID_INNE  ; XIndividadresse er
ANDNOT BIL02_INDIVID_INNE  ; XIndividadresse er
AND L2_2_AUTODREN  ; AUTODREN  L2.2
OUT 904.01
LD TR0
LD 904.01
OR=L(301) LINJEKOMMANDO &1070607
ANDLD
AND HENGER02_START  ; Xprogram starter
AND HENGER02_INDIVID_INNE  ; XIndividadresse er
ANDNOT L2_2_SPERR  ; SPERRER ALLE FUNKSJONER PAA LINJE. OGSAA VASK
SET L2_2_DRENSTART
ANDNOT P_On
SET 625.05  ; Nye drenstart L2.2
LD TR0
LD=L(301) LINJEKOMMANDO &2070607
ORNOT HENGER02_START  ; Xprogram starter
ORNOT HENGER02_INDIVID_INNE  ; XIndividadresse er
OR L2_2_SPERR  ; SPERRER ALLE FUNKSJONER PAA LINJE. OGSAA VASK
OR T0294
ANDLD
RSET L2_2_DRENSTART
RSET 625.05  ; Nye drenstart L2.2
; rung 13: MAKSTID FOR DRENERING
LD P_On
OUT TR0
AND L2_2_DRENSTART
TIM 0294 #400
LD TR0
AND T0294
OUT 635.15  ; Makstid for drenering L2.2

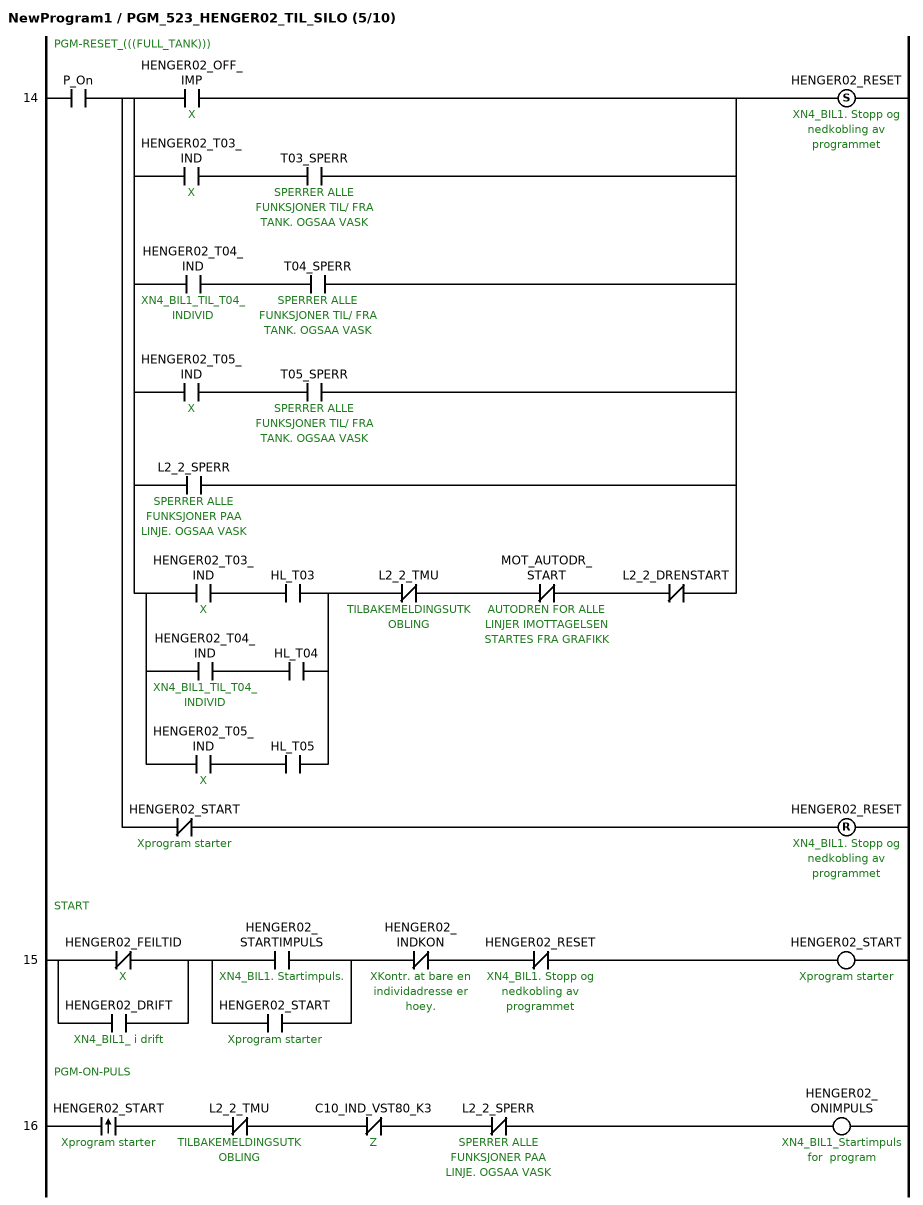
; rung 14: PGM-RESET_(((FULL_TANK)))
LD P_On
OUT TR0
LD HENGER02_OFF_IMP  ; X
LD HENGER02_T03_IND  ; X
AND T03_SPERR  ; SPERRER ALLE FUNKSJONER TIL/ FRA TANK. OGSAA VASK
ORLD
LD HENGER02_T04_IND  ; XN4_BIL1_TIL_T04_INDIVID
AND T04_SPERR  ; SPERRER ALLE FUNKSJONER TIL/ FRA TANK. OGSAA VASK
ORLD
LD HENGER02_T05_IND  ; X
AND T05_SPERR  ; SPERRER ALLE FUNKSJONER TIL/ FRA TANK. OGSAA VASK
ORLD
OR L2_2_SPERR  ; SPERRER ALLE FUNKSJONER PAA LINJE. OGSAA VASK
LD HENGER02_T03_IND  ; X
AND HL_T03
LD HENGER02_T04_IND  ; XN4_BIL1_TIL_T04_INDIVID
AND HL_T04
ORLD
LD HENGER02_T05_IND  ; X
AND HL_T05
ORLD
ANDNOT L2_2_TMU  ; TILBAKEMELDINGSUTKOBLING
ANDNOT MOT_AUTODR_START  ; AUTODREN FOR ALLE LINJER IMOTTAGELSEN STARTES FRA GRAFIKK
ANDNOT L2_2_DRENSTART
ORLD
ANDLD
SET HENGER02_RESET  ; XN4_BIL1. Stopp og nedkobling av programmet
LD TR0
ANDNOT HENGER02_START  ; Xprogram starter
RSET HENGER02_RESET  ; XN4_BIL1. Stopp og nedkobling av programmet
; rung 15: START
LDNOT HENGER02_FEILTID  ; X
OR HENGER02_DRIFT  ; XN4_BIL1_ i drift
LD HENGER02_STARTIMPULS  ; XN4_BIL1. Startimpuls.
OR HENGER02_START  ; Xprogram starter
ANDLD
ANDNOT HENGER02_INDKON  ; XKontr. at bare en individadresse er hoey.
ANDNOT HENGER02_RESET  ; XN4_BIL1. Stopp og nedkobling av programmet
OUT HENGER02_START  ; Xprogram starter
; rung 16: PGM-ON-PULS
@LD HENGER02_START  ; Xprogram starter
ANDNOT L2_2_TMU  ; TILBAKEMELDINGSUTKOBLING
ANDNOT C10_IND_VST80_K3  ; Z
ANDNOT L2_2_SPERR  ; SPERRER ALLE FUNKSJONER PAA LINJE. OGSAA VASK
OUT HENGER02_ONIMPULS  ; XN4_BIL1_Startimpuls for  program

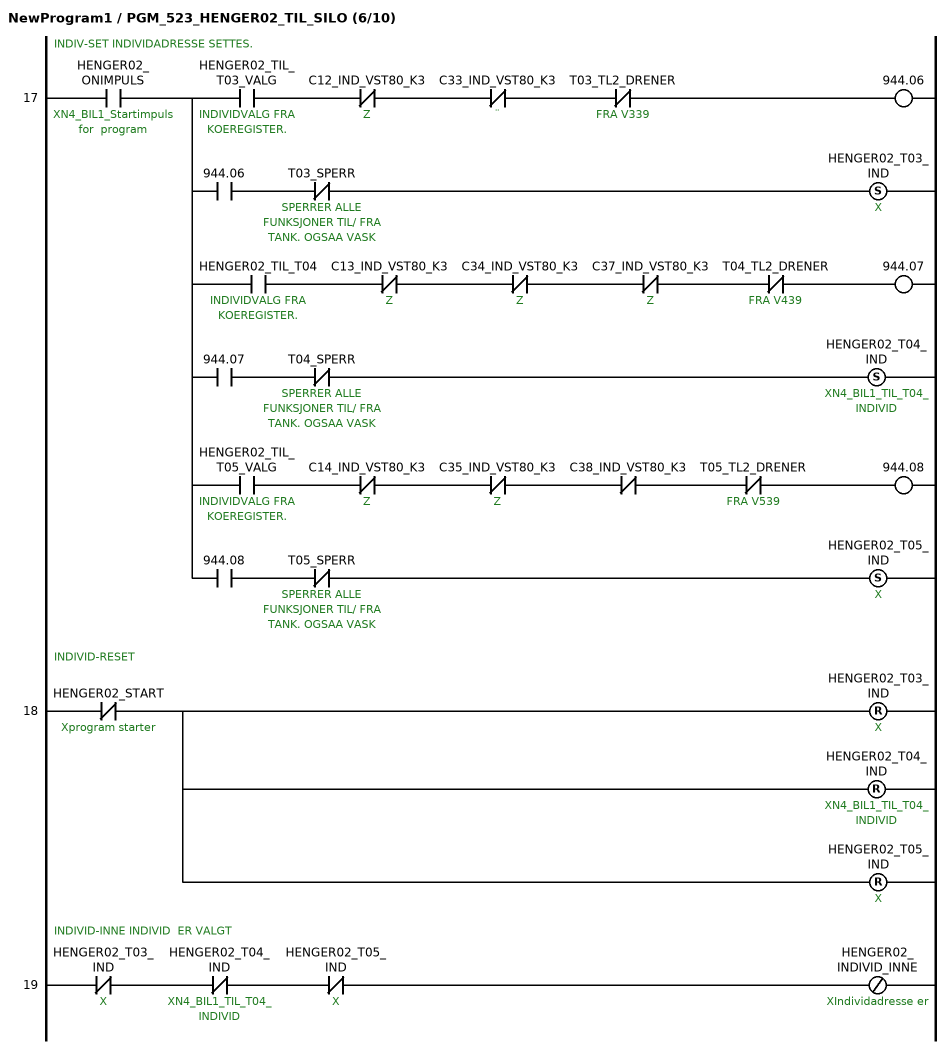
; rung 17: INDIV-SET INDIVIDADRESSE SETTES.
LD HENGER02_ONIMPULS  ; XN4_BIL1_Startimpuls for  program
OUT TR0
AND HENGER02_TIL_T03_VALG  ; INDIVIDVALG FRA KOEREGISTER.
ANDNOT C12_IND_VST80_K3  ; Z
ANDNOT C33_IND_VST80_K3  ; ¨
ANDNOT T03_TL2_DRENER  ; FRA V339
OUT 944.06
LD TR0
AND 944.06
ANDNOT T03_SPERR  ; SPERRER ALLE FUNKSJONER TIL/ FRA TANK. OGSAA VASK
SET HENGER02_T03_IND  ; X
LD TR0
AND HENGER02_TIL_T04  ; INDIVIDVALG FRA KOEREGISTER.
ANDNOT C13_IND_VST80_K3  ; Z
ANDNOT C34_IND_VST80_K3  ; Z
ANDNOT C37_IND_VST80_K3  ; Z
ANDNOT T04_TL2_DRENER  ; FRA V439
OUT 944.07
LD TR0
AND 944.07
ANDNOT T04_SPERR  ; SPERRER ALLE FUNKSJONER TIL/ FRA TANK. OGSAA VASK
SET HENGER02_T04_IND  ; XN4_BIL1_TIL_T04_INDIVID
LD TR0
AND HENGER02_TIL_T05_VALG  ; INDIVIDVALG FRA KOEREGISTER.
ANDNOT C14_IND_VST80_K3  ; Z
ANDNOT C35_IND_VST80_K3  ; Z
ANDNOT C38_IND_VST80_K3
ANDNOT T05_TL2_DRENER  ; FRA V539
OUT 944.08
LD TR0
AND 944.08
ANDNOT T05_SPERR  ; SPERRER ALLE FUNKSJONER TIL/ FRA TANK. OGSAA VASK
SET HENGER02_T05_IND  ; X
; rung 18: INDIVID-RESET
LDNOT HENGER02_START  ; Xprogram starter
RSET HENGER02_T03_IND  ; X
RSET HENGER02_T04_IND  ; XN4_BIL1_TIL_T04_INDIVID
RSET HENGER02_T05_IND  ; X
; rung 19: INDIVID-INNE INDIVID  ER VALGT
LDNOT HENGER02_T03_IND  ; X
ANDNOT HENGER02_T04_IND  ; XN4_BIL1_TIL_T04_INDIVID
ANDNOT HENGER02_T05_IND  ; X
OUTNOT HENGER02_INDIVID_INNE  ; XIndividadresse er

